SUBAPPLICATION Luftventil (* Steuert den digitalen Ausgang (MI_00 / DigitalOutput_2A) fuer das Luftventil und meldet dessen Ist-Zustand sowie Status zurueck *)
  (* Standard: 61499-2 *)
  (* Version 1.0, 2024-04-23, Elias *)
  IMPORT DataPanel::io::MI::DQ::DataPanel_MI_DO::DigitalOutput_2A;
  IMPORT DataPanel::io::MI::const::MI::MI_00;
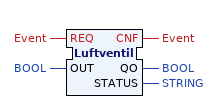
  EVENT_INPUT
    REQ; (* Anforderung: Ausgang gemaess OUT ansteuern *)
  END_EVENT
  EVENT_OUTPUT
    CNF; (* Bestaetigung: Ansteuerung abgeschlossen *)
  END_EVENT
  VAR_INPUT
    OUT : BOOL; (* Sollwert des Ausgangs (TRUE = Luftventil geoeffnet) *)
  END_VAR
  VAR_OUTPUT
    QO : BOOL; (* Rueckgelesener Ist-Zustand des digitalen Ausgangs *)
    STATUS : STRING; (* Status-/Diagnosemeldung des digitalen Ausgangs *)
  END_VAR
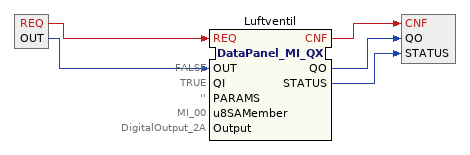
  FBS
    Luftventil : DataPanel::io::MI::DQ::DataPanel_MI_QX(QI := TRUE, PARAMS := '', OUT := FALSE, u8SAMember := MI_00, Output := DigitalOutput_2A);
  END_FBS
  EVENT_CONNECTIONS
    REQ TO Luftventil.REQ;
    Luftventil.CNF TO CNF;
  END_CONNECTIONS
  DATA_CONNECTIONS
    OUT TO Luftventil.OUT;
    Luftventil.QO TO QO;
    Luftventil.STATUS TO STATUS;
  END_CONNECTIONS
END_SUBAPPLICATION
